(* PLC project ramp_1dir_2speed, Dassault Systèmes ControlBuild 2024x *)
(* stored: creationDateTime 2023-10-03T11:13:18-01:00 *)

(* This module simulates the behaviour of a bounded ramp according to the state of 2 boolean inputs. *)
FUNCTION_BLOCK equipment_library.ramp_1dir_2speed
  VAR_INPUT
    fwdHighSpeedState : BOOL := false;
    fwdLowSpeedState : BOOL := false;
  END_VAR
  VAR_OUTPUT
    positionRamp : REAL := 0.0;
    percentRamp : REAL := 0.0;
  END_VAR
  VAR
    increment : REAL := 0.0;
    pBound : REAL := 0.0;
  END_VAR
  VAR CONSTANT
    maxRamp : REAL := 1000.0;
    timeRamp : REAL := 10.0;
  END_VAR
  VAR
    d_locking : BOOL := false;
    v_d_locking : REAL := 10.0;
  END_VAR


ACTION C_source_code:
/* ----------------------------------------------------------------	*/
/* Type : Model of Operative Behaviour					*/
/* Category :  Actuators							*/
/* Author : Dassault Systemes						*/
/* Update date : June 2018							*/
/* ----------------------------------------------------------------	*/
/* This module simulates the behaviour of a bounded ramp according	*/
/* to the state of 2 boolean inputs.					*/
/* ----------------------------------------------------------------	*/


/* ----------------------------------------------------------------	*/
/* Compute the ramp								*/
/* ----------------------------------------------------------------	*/
if (! d_locking)  {
	/* Compute the increment of translation according to the simulation clock	*/
	if (timeRamp > 0.0)
			increment=(maxRamp/timeRamp)*(CLOCK_PERIOD/1000000.0);

	/* Compute the target according to inputs	*/
	if (fwdHighSpeedState) pBound = maxRamp;
	else if (fwdLowSpeedState) {
		pBound = maxRamp / 2.0;
		increment = increment / 2.0;
	}
	if (! fwdHighSpeedState && ! fwdLowSpeedState) pBound = 0.0;

	/* Compute the value of the ramp	*/
	if ( positionRamp < pBound ) {
		positionRamp += increment;
		if ( positionRamp > pBound ) positionRamp = pBound;
	}
	if ( positionRamp > pBound ) {
		positionRamp -= increment;
		if (positionRamp < pBound) positionRamp = pBound;
	}
}



/* ----------------------------------------------------------------	*/
/* Compute the percentage of the height of the ramp			*/
/* ----------------------------------------------------------------	*/
if (maxRamp > 0.0)
	percentRamp = ((positionRamp/maxRamp)*100);
END_ACTION
END_FUNCTION_BLOCK
